(* IEC 61131-3 sources: repolevel_ST_code_completion/extract_code/三轴CNC运动实训/FUN, 5 files *)

(* ---- INIT_CNC_System.st ---- *)
FUNCTION INIT_CNC_System : BOOL
VAR_IN_OUT
	fbSMC_ReadNCFile		:	SMC_ReadNCFile;
	fbSMC_NCDecoder			:	SMC_NCDecoder;
	fbSMC_CheckVelocities	:	SMC_CheckVelocities;
	fbSMC_Interpolator		:	SMC_Interpolator;
	fbSMC_ControlAxisXByPos	:	SMC_ControlAxisByPos;
	fbSMC_ControlAxisYByPos	:	SMC_ControlAxisByPos;
	fbSMC_ControlAxisZByPos	:	SMC_ControlAxisByPos;
	fbSMC_AXISX_HOMING		:	SMC_HOMING;
	fbSMC_AXISY_HOMING		:	SMC_HOMING;
	fbSMC_AXISZ_HOMING		:	SMC_HOMING;
	fbMC_AXISX_STOP			:	MC_STOP;
	fbMC_AXISY_STOP			:	MC_STOP;
	fbMC_AXISZ_STOP			:	MC_STOP;
END_VAR
VAR_INPUT
	AxisX					:	SM3_Basic.AXIS_REF_SM3
	AxisY					:	SM3_Basic.AXIS_REF_SM3
	AxisZ					:	SM3_Basic.AXIS_REF_SM3
END_VAR

// 复位回零标志
// 注意：这里不能直接修改VAR_INPUT的变量，需要在调用处理

// 复位G代码处理相关功能块
fbSMC_ReadNCFile(bExecute := FALSE);
fbSMC_NCDecoder(bExecute := FALSE, ncprog := fbSMC_ReadNCFile.ncprog);
fbSMC_CheckVelocities(bExecute := FALSE);
fbSMC_Interpolator(bExecute := FALSE);

// 复位轴控制功能块
fbSMC_ControlAxisXByPos(bEnable := FALSE, Axis := AxisX);
fbSMC_ControlAxisYByPos(bEnable := FALSE, Axis := AxisY);
fbSMC_ControlAxisZByPos(bEnable := FALSE, Axis := AxisZ);

// 复位回零功能块
fbSMC_AXISX_HOMING(bExecute := FALSE, Axis := AxisX);
fbSMC_AXISY_HOMING(bExecute := FALSE, Axis := AxisY);
fbSMC_AXISZ_HOMING(bExecute := FALSE, Axis := AxisZ);

// 复位停止功能块
fbMC_AXISX_STOP(Execute := FALSE, Deceleration := 100, Axis := AxisX);
fbMC_AXISY_STOP(Execute := FALSE, Deceleration := 100, Axis := AxisY);
fbMC_AXISZ_STOP(Execute := FALSE, Deceleration := 100, Axis := AxisZ);

// 返回TRUE表示初始化完成
INIT_CNC_System := TRUE;

(* ---- FB_TripleAxisHoming.st ---- *)
FUNCTION_BLOCK FB_TripleAxisHoming
VAR_INPUT
	bExecute			:	BOOL;				//执行回零信号
	AxisX				:	SM3_Basic.AXIS_REF_SM3;			//X轴引用
	AxisY				:	SM3_Basic.AXIS_REF_SM3;			//Y轴引用
	AxisZ				:	SM3_Basic.AXIS_REF_SM3;			//Z轴引用
	bAxisXRefSwitch		:	BOOL;				//X轴零点开关
	bAxisYRefSwitch		:	BOOL;				//Y轴零点开关
	bAxisZRefSwitch		:	BOOL;				//Z轴零点开关
	fVelocitySlow		:	REAL;				//慢速回零速度
	fVelocityFast		:	REAL;				//快速回零速度
	fAcceleration		:	REAL;				//加速度
	fDeceleration		:	REAL;				//减速度
END_VAR
VAR_OUTPUT
	bHomeOK				:	BOOL;				//三轴都回零完成
	bAxisXHomeOK		:	BOOL;				//X轴回零完成
	bAxisYHomeOK		:	BOOL;				//Y轴回零完成
	bAxisZHomeOK		:	BOOL;				//Z轴回零完成
	bBusy				:	BOOL;				//回零进行中
	bError				:	BOOL;				//错误标志
	sErrorString		:	STRING;				//错误信息字符串
END_VAR
VAR
	fbHomingX			:	SMC_HOMING;			//X轴回零功能块
	fbHomingY			:	SMC_HOMING;			//Y轴回零功能块
	fbHomingZ			:	SMC_HOMING;			//Z轴回零功能块
	fbDoneXTrig			:	R_TRIG;				//X轴完成上升沿
	fbDoneYTrig			:	R_TRIG;				//Y轴完成上升沿
	fbDoneZTrig			:	R_TRIG;				//Z轴完成上升沿
END_VAR

// X轴回零
fbHomingX(
	bExecute := bExecute,
	bReferenceSwitch := bAxisXRefSwitch,
	fVelocitySlow := fVelocitySlow,
	fVelocityFast := fVelocityFast,
	fAcceleration := fAcceleration,
	fDeceleration := fDeceleration,
	Axis := AxisX
);

// Y轴回零
fbHomingY(
	bExecute := bExecute,
	bReferenceSwitch := bAxisYRefSwitch,
	fVelocitySlow := fVelocitySlow,
	fVelocityFast := fVelocityFast,
	fAcceleration := fAcceleration,
	fDeceleration := fDeceleration,
	Axis := AxisY
);

// Z轴回零
fbHomingZ(
	bExecute := bExecute,
	bReferenceSwitch := bAxisZRefSwitch,
	fVelocitySlow := fVelocitySlow,
	fVelocityFast := fVelocityFast,
	fAcceleration := fAcceleration,
	fDeceleration := fDeceleration,
	Axis := AxisZ
);

// 检测X轴完成
fbDoneXTrig(CLK := fbHomingX.bDone);
IF fbDoneXTrig.Q THEN
	bAxisXHomeOK := TRUE;
END_IF

// 检测Y轴完成
fbDoneYTrig(CLK := fbHomingY.bDone);
IF fbDoneYTrig.Q THEN
	bAxisYHomeOK := TRUE;
END_IF

// 检测Z轴完成
fbDoneZTrig(CLK := fbHomingZ.bDone);
IF fbDoneZTrig.Q THEN
	bAxisZHomeOK := TRUE;
END_IF

// 更新输出状态
bHomeOK := bAxisXHomeOK AND bAxisYHomeOK AND bAxisZHomeOK;
bBusy := fbHomingX.bBusy OR fbHomingY.bBusy OR fbHomingZ.bBusy;

// 错误检查（优先级：X > Y > Z）
IF fbHomingX.bError THEN
	bError := TRUE;
	SMC_ERRORSTRING(ErrorID := fbHomingX.nErrorID, Language := english, SMC_ErrorString => sErrorString);
ELSIF fbHomingY.bError THEN
	bError := TRUE;
	SMC_ERRORSTRING(ErrorID := fbHomingY.nErrorID, Language := english, SMC_ErrorString => sErrorString);
ELSIF fbHomingZ.bError THEN
	bError := TRUE;
	SMC_ERRORSTRING(ErrorID := fbHomingZ.nErrorID, Language := english, SMC_ErrorString => sErrorString);
ELSE
	bError := FALSE;
	sErrorString := 'CNC_NO_ERROR';
END_IF

// 复位逻辑
IF NOT bExecute THEN
	bAxisXHomeOK := FALSE;
	bAxisYHomeOK := FALSE;
	bAxisZHomeOK := FALSE;
	bHomeOK := FALSE;
END_IF

(* ---- FB_TripleAxisPower.st ---- *)
FUNCTION_BLOCK FB_TripleAxisPower
VAR_INPUT
	AxisX			:	SM3_Basic.AXIS_REF_SM3			//X轴引用
	AxisY			:	SM3_Basic.AXIS_REF_SM3			//Y轴引用
	AxisZ			:	SM3_Basic.AXIS_REF_SM3			//Z轴引用
	bServoEnable	:	BOOL;				//伺服使能信号
END_VAR
VAR_OUTPUT
	bReady			:	BOOL;				//三轴都准备就绪
	bAxisXReady		:	BOOL;				//X轴准备就绪
	bAxisYReady		:	BOOL;				//Y轴准备就绪
	bAxisZReady		:	BOOL;				//Z轴准备就绪
	bError			:	BOOL;				//错误标志
	sErrorString	:	STRING;				//错误信息字符串
END_VAR
VAR
	fbPowerX		:	MC_POWER;			//X轴电源控制
	fbPowerY		:	MC_POWER;			//Y轴电源控制
	fbPowerZ		:	MC_POWER;			//Z轴电源控制
END_VAR

// X轴电源控制
fbPowerX(
	Enable := bServoEnable,
	bRegulatorOn := bServoEnable,
	bDriveStart := bServoEnable,
	Axis := AxisX
);

// Y轴电源控制
fbPowerY(
	Enable := bServoEnable,
	bRegulatorOn := bServoEnable,
	bDriveStart := bServoEnable,
	Axis := AxisY
);

// Z轴电源控制
fbPowerZ(
	Enable := bServoEnable,
	bRegulatorOn := bServoEnable,
	bDriveStart := bServoEnable,
	Axis := AxisZ
);

// 更新输出状态
bAxisXReady := fbPowerX.Status;
bAxisYReady := fbPowerY.Status;
bAxisZReady := fbPowerZ.Status;
bReady := fbPowerX.Status AND fbPowerY.Status AND fbPowerZ.Status;

// 错误检查（优先级：X > Y > Z）
IF fbPowerX.Error THEN
	bError := TRUE;
	SMC_ERRORSTRING(ErrorID := fbPowerX.ErrorID, Language := english, SMC_ErrorString => sErrorString);
ELSIF fbPowerY.Error THEN
	bError := TRUE;
	SMC_ERRORSTRING(ErrorID := fbPowerY.ErrorID, Language := english, SMC_ErrorString => sErrorString);
ELSIF fbPowerZ.Error THEN
	bError := TRUE;
	SMC_ERRORSTRING(ErrorID := fbPowerZ.ErrorID, Language := english, SMC_ErrorString => sErrorString);
ELSE
	bError := FALSE;
	sErrorString := 'CNC_NO_ERROR';
END_IF

(* ---- FB_TripleAxisReset.st ---- *)
FUNCTION_BLOCK FB_TripleAxisReset
VAR_INPUT
	AxisX			:	SM3_Basic.AXIS_REF_SM3			//X轴引用
	AxisY			:	SM3_Basic.AXIS_REF_SM3			//Y轴引用
	AxisZ			:	SM3_Basic.AXIS_REF_SM3			//Z轴引用
	bExecute		:	BOOL;				//执行复位信号
END_VAR
VAR_OUTPUT
	bDone			:	BOOL;				//三轴都复位完成
	bBusy			:	BOOL;				//复位进行中
	bError			:	BOOL;				//错误标志
	sErrorString	:	STRING;				//错误信息字符串
END_VAR
VAR
	fbResetX		:	MC_RESET;			//X轴复位
	fbResetY		:	MC_RESET;			//Y轴复位
	fbResetZ		:	MC_RESET;			//Z轴复位
END_VAR

// X轴复位
fbResetX(
	Execute := bExecute,
	Axis := AxisX
);

// Y轴复位
fbResetY(
	Execute := bExecute,
	Axis := AxisY
);

// Z轴复位
fbResetZ(
	Execute := bExecute,
	Axis := AxisZ
);

// 更新输出状态
bBusy := fbResetX.Busy OR fbResetY.Busy OR fbResetZ.Busy;
bDone := fbResetX.Done AND fbResetY.Done AND fbResetZ.Done;

// 错误检查（优先级：X > Y > Z）
IF fbResetX.Error THEN
	bError := TRUE;
	SMC_ERRORSTRING(ErrorID := fbResetX.ErrorID, Language := english, SMC_ErrorString => sErrorString);
ELSIF fbResetY.Error THEN
	bError := TRUE;
	SMC_ERRORSTRING(ErrorID := fbResetY.ErrorID, Language := english, SMC_ErrorString => sErrorString);
ELSIF fbResetZ.Error THEN
	bError := TRUE;
	SMC_ERRORSTRING(ErrorID := fbResetZ.ErrorID, Language := english, SMC_ErrorString => sErrorString);
ELSE
	bError := FALSE;
	sErrorString := 'CNC_NO_ERROR';
END_IF

(* ---- FB_TripleAxisStop.st ---- *)
FUNCTION_BLOCK FB_TripleAxisStop
VAR_INPUT
	AxisX			:	SM3_Basic.AXIS_REF_SM3			//X轴引用
	AxisY			:	SM3_Basic.AXIS_REF_SM3			//Y轴引用
	AxisZ			:	SM3_Basic.AXIS_REF_SM3			//Z轴引用
	bExecute		:	BOOL;				//执行停止信号
	rDeceleration	:	REAL := 100.0;		//减速度
END_VAR
VAR_OUTPUT
	bDone			:	BOOL;				//三轴都停止完成
	bBusy			:	BOOL;				//停止进行中
	bError			:	BOOL;				//错误标志
	sErrorString	:	STRING;				//错误信息字符串
END_VAR
VAR
	fbStopX			:	MC_STOP;			//X轴停止
	fbStopY			:	MC_STOP;			//Y轴停止
	fbStopZ			:	MC_STOP;			//Z轴停止
END_VAR

// X轴停止
fbStopX(
	Execute := bExecute,
	Deceleration := rDeceleration,
	Axis := AxisX
);

// Y轴停止
fbStopY(
	Execute := bExecute,
	Deceleration := rDeceleration,
	Axis := AxisY
);

// Z轴停止
fbStopZ(
	Execute := bExecute,
	Deceleration := rDeceleration,
	Axis := AxisZ
);

// 更新输出状态
bBusy := fbStopX.Busy OR fbStopY.Busy OR fbStopZ.Busy;
bDone := fbStopX.Done AND fbStopY.Done AND fbStopZ.Done;

// 错误检查（优先级：X > Y > Z）
IF fbStopX.Error THEN
	bError := TRUE;
	SMC_ERRORSTRING(ErrorID := fbStopX.ErrorID, Language := english, SMC_ErrorString => sErrorString);
ELSIF fbStopY.Error THEN
	bError := TRUE;
	SMC_ERRORSTRING(ErrorID := fbStopY.ErrorID, Language := english, SMC_ErrorString => sErrorString);
ELSIF fbStopZ.Error THEN
	bError := TRUE;
	SMC_ERRORSTRING(ErrorID := fbStopZ.ErrorID, Language := english, SMC_ErrorString => sErrorString);
ELSE
	bError := FALSE;
	sErrorString := 'CNC_NO_ERROR';
END_IF
